PROGRAM example_loop_control
VAR

END_VAR

// NETWORK 1

END_PROGRAM

(* stored: Version 1.1.0.1, ProductVersion 3.1.4024.12
   POU example_loop_control: Id {f4111f27-f002-47e1-985a-deb6fca944d4}, SpecialFunc None *)
